PROGRAM V0_2
VAR
END_VAR

(*
	Twee signalen
	
	Als S01=1 en S02=0 moet Q01 branden
	Als S01=0 en S02=1 moet Q02 branden
	Als S01=0 en S02=0 moet Q01 en Q02 branden
	Als S01=1 en S02=1 moet Q01 en Q02 niet branden
	
	S1	S2	Q1	Q2
	0	0	1	1
	0	1	0	1
	1	0	1	0
	1	1	0	0
*)

GVL.bLamp_1 := (NOT GVL.bSwitch_2);
GVL.bLamp_2 := (NOT GVL.bSwitch_1);

END_PROGRAM

(* stored: Version 1.1.0.1, ProductVersion 3.1.4024.12
   POU V0_2: Id {b6d42e48-56aa-49b2-8505-3dcae3a33928}, SpecialFunc None *)
